FUNCTION SaveNewBinPosition
VAR_INPUT
END_VAR
VAR
END_VAR

//New position of bin1
IF MeasuringData.SaveNewPositionOfBin1 THEN
	MeasuringData.Bin1Position := MAIN.AxisControl.ActualPosition;
END_IF
//New position of bin2
IF MeasuringData.SaveNewPositionOfBin2 THEN
	MeasuringData.Bin2Position := MAIN.AxisControl.ActualPosition;
END_IF
//New position of bin3
IF MeasuringData.SaveNewPositionOfBin3 THEN
	MeasuringData.Bin3Position := MAIN.AxisControl.ActualPosition;
END_IF
//New position of bin4
IF MeasuringData.SaveNewPositionOfBin4 THEN
	MeasuringData.Bin4Position := MAIN.AxisControl.ActualPosition;
END_IF

END_FUNCTION

(* stored: Version 1.1.0.1, ProductVersion 3.1.4024.13
   POU SaveNewBinPosition: Id {3e015298-61f8-4e0a-a10f-f01c34e186b9}, SpecialFunc None *)
